// TIA Portal V20 export
DATA_BLOCK "Config"   // DB69
// stored: MemoryReserve 100, Namespace Unit1.Em7
   VAR
      em : "LAF_typeEmConfiguration";   // Configuration of EM Parameters
      cmHotPressRightSafetyPin : "LBC_typeDigitalSignalConfiguration";
      cmHotPressRightJRDetect : "LBC_typeDigitalSignalConfiguration";
      cmHotPressRightStageLiftFrontUpDown : "LBC_typeTwoWayActuatorConfiguration";
      cmHotPressRightStageLiftRearUpDown : "LBC_typeTwoWayActuatorConfiguration";
      cmHotPressRightStageLiftAllUpDown : "LBC_typeTwoWayActuatorConfiguration";
      cmHotPressRightServoPress : "LER_typeServoPressConfiguration";
      cmHotPressRightTemperature : "LER_typeHeaterConfiguration";
   END_VAR
BEGIN
   em.referenceDesignator.parent := WSTRING#'U1';
   em.referenceDesignator.relative := WSTRING#'EM0';
   cmHotPressRightStageLiftFrontUpDown.referenceDesignator := WSTRING#'HP STAGE LIFT FRONT';
   cmHotPressRightStageLiftFrontUpDown.monitoringDiscrepancy := T#5s;
   cmHotPressRightStageLiftRearUpDown.referenceDesignator := WSTRING#'HP STAGE LIFT REAR';
   cmHotPressRightStageLiftRearUpDown.monitoringDiscrepancy := T#5s;
   cmHotPressRightStageLiftAllUpDown.referenceDesignator := WSTRING#'Stage';
   cmHotPressRightStageLiftAllUpDown.monitoringDiscrepancy := T#5s;
   cmHotPressRightServoPress.hwID."220ByteIn" := 652;
   cmHotPressRightServoPress.hwID."220ByteOut" := 651;
   cmHotPressRightTemperature.MB_Comm_Load.PORT := 1056;
   cmHotPressRightTemperature.MB_Comm_Load.BAUD := 9600;
   cmHotPressRightTemperature.MB_Comm_Load.PARITY := 2;
END_DATA_BLOCK
